FUNCTION_BLOCK SemephoreV1
VAR_INPUT
	currentMode : eOperationModes;
	isError : BOOL;
	isInitializing : BOOL;
END_VAR
VAR_OUTPUT
END_VAR
VAR
	io : POINTER TO ioBundleControl;
	buzzerCounter : INT;
END_VAR
VAR PERSISTENT
	buzzerTimerOn : TON;
	buzzerTimerOff : TON;
	buzzerGoal : INT := 5;
	buzzerEnable : bool := false;
END_VAR

//reset all
io^.lightGreen := FALSE;
io^.lightRed := FALSE;
io^.lightYellow := FALSE;
io^.lightWhite := FALSE;
io^.towerGreen := FALSE;
io^.towerRed := FALSE;
io^.towerYellow := FALSE;
//io^.towerBuzzer := FALSE;

CASE currentMode OF
	eOperationModes.AUTO:
		io^.lightGreen := TRUE;
	eOperationModes.MANUAL,eOperationModes.SEMI_AUTO:
		io^.lightRed := TRUE;
		io^.towerYellow := TRUE;
END_CASE

io^.lightYellow := isError OR isInitializing;
io^.towerRed := isError;
io^.towerYellow := io^.towerYellow OR isInitializing;
io^.towerGreen := NOT io^.towerRed AND NOT io^.towerYellow;

//buzser (fliper
buzzerTimerOn(IN:= , PT:= , Q=>, ET=> );
buzzerTimerOff(IN:= , PT:= , Q=> , ET=> );

IF buzzerTimerOn.Q THEN
	buzzerTimerOff.IN := TRUE;
	buzzerTimerOn.IN := FALSE;
ELSIF buzzerTimerOff.Q THEN
	buzzerTimerOff.IN := FALSE;
	buzzerTimerOn.IN := TRUE;
	
	buzzerCounter := buzzerCounter +1; // a cycle complished
	
ELSIF NOT buzzerTimerOn.IN AND NOT buzzerTimerOff.IN THEN
	buzzerTimerOn.IN := TRUE;
END_IF

IF  NOT isError THEN
	buzzerCounter := 0;
END_IF
// error comes and timeron and counter not reached
io^.towerBuzzer := isError AND buzzerTimerOn.Q AND (buzzerCounter < buzzerGoal) and buzzerEnable;

METHOD FB_init : BOOL
VAR_INPUT
	bInitRetains : BOOL; // if TRUE, the retain variables are initialized (warm start / cold start)
	bInCopyCode : BOOL;  // if TRUE, the instance afterwards gets moved into the copy code (online change)
	
	argIo : pointer to ioBundleControl;
END_VAR
io := argIo;
END_METHOD

END_FUNCTION_BLOCK

(* stored: Version 1.1.0.1, ProductVersion 3.1.4024.0
   POU SemephoreV1: Id {c757335b-0259-4bad-9739-4559055a1f86}, SpecialFunc None
   Method FB_init: Id {5d97e876-0d51-4c4d-9ca6-9c927dbc5548} *)
